# EPICS substitutions: db/ecmcEL3632_s5.substitutions
file ecmcEcSlave.template
{
    pattern {}
            {}
}

file ecmcEL3632-chX.template
{
	pattern {CH_ID, DTYP,             FTVL,  NELM}
		    {1,     asynInt16ArrayIn, SHORT, 5   }
		    {2,     asynInt16ArrayIn, SHORT, 5   }
}
